FUNCTION_BLOCK RegisterServiceOpcUa (* Register Service using OPC UA *)
  (* Standard: 61499-2; Description: Copyright (c) 2019 fortiss GmbH This program and the accompanying materials are made available under the terms of the Eclipse Public License 2.0 which is available at https://www.eclipse.org/legal/epl-2.0/ SPDX-License-Identifier: EPL-2.0 *)
  (* Version 1.0, 2019-09-17, Jose Cabral, fortiss GmbH *)
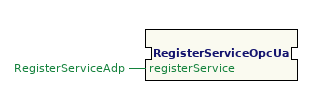
  SOCKETS
    registerService : RegisterServiceAdp; (* Register Service adapter *)
  END_SOCKETS
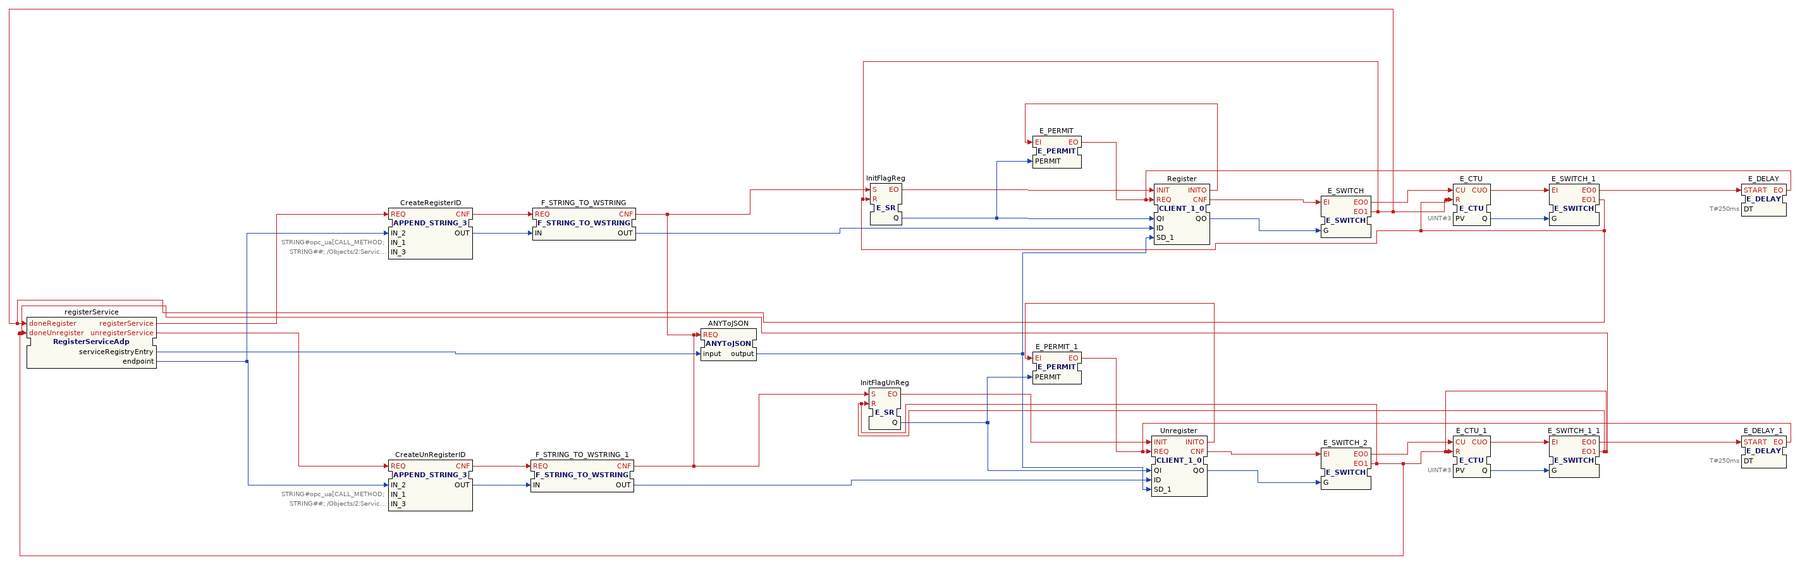
  FBS
    InitFlagReg : E_SR;
    E_PERMIT : E_PERMIT;
    CreateRegisterID : APPEND_STRING_3(IN_1 := STRING#opc_ua[CALL_METHOD; , IN_3 := STRING##; /Objects/2:ServiceRegistry/2:register]);
    F_STRING_TO_WSTRING : F_STRING_TO_WSTRING;
    E_PERMIT_1 : E_PERMIT;
    InitFlagUnReg : E_SR;
    CreateUnRegisterID : APPEND_STRING_3(IN_1 := STRING#opc_ua[CALL_METHOD; , IN_3 := STRING##; /Objects/2:ServiceRegistry/2:remove]);
    F_STRING_TO_WSTRING_1 : F_STRING_TO_WSTRING;
    ANYToJSON : ANYToJSON;
    Register : CLIENT_1_0;
    Unregister : CLIENT_1_0;
    E_SWITCH : E_SWITCH;
    E_SWITCH_1 : E_SWITCH;
    E_DELAY : E_DELAY(DT := T#250ms);
    E_CTU : E_CTU(PV := UINT#3);
    E_SWITCH_1_1 : E_SWITCH;
    E_SWITCH_2 : E_SWITCH;
    E_DELAY_1 : E_DELAY(DT := T#250ms);
    E_CTU_1 : E_CTU(PV := UINT#3);
  END_FBS
  EVENT_CONNECTIONS
    CreateRegisterID.CNF TO F_STRING_TO_WSTRING.REQ;
    F_STRING_TO_WSTRING.CNF TO InitFlagReg.S;
    CreateUnRegisterID.CNF TO F_STRING_TO_WSTRING_1.REQ;
    F_STRING_TO_WSTRING_1.CNF TO InitFlagUnReg.S;
    F_STRING_TO_WSTRING.CNF TO ANYToJSON.REQ;
    F_STRING_TO_WSTRING_1.CNF TO ANYToJSON.REQ;
    registerService.registerService TO CreateRegisterID.REQ;
    registerService.unregisterService TO CreateUnRegisterID.REQ;
    InitFlagReg.EO TO Register.INIT;
    E_PERMIT.EO TO Register.REQ;
    Register.INITO TO E_PERMIT.EI;
    InitFlagUnReg.EO TO Unregister.INIT;
    E_PERMIT_1.EO TO Unregister.REQ;
    Unregister.INITO TO E_PERMIT_1.EI;
    E_CTU.CUO TO E_SWITCH_1.EI;
    E_SWITCH_1.EO0 TO E_DELAY.START;
    E_SWITCH.EO0 TO E_CTU.CU;
    E_SWITCH.EO1 TO InitFlagReg.R;
    E_SWITCH.EO1 TO registerService.doneRegister;
    Register.CNF TO E_SWITCH.EI;
    E_DELAY.EO TO Register.REQ;
    E_SWITCH_1_1.EO0 TO E_DELAY_1.START;
    E_CTU_1.CUO TO E_SWITCH_1_1.EI;
    E_SWITCH_2.EO0 TO E_CTU_1.CU;
    E_SWITCH_2.EO1 TO InitFlagUnReg.R;
    E_SWITCH_2.EO1 TO registerService.doneUnregister;
    Unregister.CNF TO E_SWITCH_2.EI;
    E_DELAY_1.EO TO Unregister.REQ;
    E_SWITCH_1_1.EO1 TO InitFlagUnReg.R;
    E_SWITCH_1.EO1 TO InitFlagReg.R;
    E_SWITCH_1_1.EO1 TO registerService.doneUnregister;
    E_SWITCH_1.EO1 TO registerService.doneRegister;
    E_SWITCH_1_1.EO1 TO E_CTU_1.R;
    E_SWITCH_2.EO1 TO E_CTU_1.R;
    E_SWITCH.EO1 TO E_CTU.R;
    E_SWITCH_1.EO1 TO E_CTU.R;
  END_CONNECTIONS
  DATA_CONNECTIONS
    InitFlagReg.Q TO E_PERMIT.PERMIT;
    CreateRegisterID.OUT TO F_STRING_TO_WSTRING.IN;
    CreateUnRegisterID.OUT TO F_STRING_TO_WSTRING_1.IN;
    InitFlagUnReg.Q TO E_PERMIT_1.PERMIT;
    registerService.serviceRegistryEntry TO ANYToJSON.input;
    registerService.endpoint TO CreateRegisterID.IN_2;
    registerService.endpoint TO CreateUnRegisterID.IN_2;
    InitFlagReg.Q TO Register.QI;
    F_STRING_TO_WSTRING.OUT TO Register.ID;
    ANYToJSON.output TO Register.SD_1;
    InitFlagUnReg.Q TO Unregister.QI;
    F_STRING_TO_WSTRING_1.OUT TO Unregister.ID;
    ANYToJSON.output TO Unregister.SD_1;
    E_CTU.Q TO E_SWITCH_1.G;
    Register.QO TO E_SWITCH.G;
    E_CTU_1.Q TO E_SWITCH_1_1.G;
    Unregister.QO TO E_SWITCH_2.G;
  END_CONNECTIONS
END_FUNCTION_BLOCK
